(* PLC project Adressering.ecp, WAGO e!COCKPIT e!COCKPIT *)
(* stored: creationDateTime 2021-01-18T14:20:23.2110188, modificationDateTime 2021-01-18T11:51:27.6823754 *)

TYPE dtRomtype_112 : STRUCT
  RB601_V : BOOL;  (* Bevegelse *)
  RB601_HVAC : BOOL;  (* HVAC signal *)
  RT601_CT : REAL;  (* Rom temperatur *)
  RT602_CT : REAL;  (* Rom temperatur *)
  RT602_SP : REAL;  (* Temperatur SP *)
  RT601_SP_D : REAL;  (* Temperatur SP *)
  RT601_SP_S : REAL;  (* Temperatur SP standby *)
  RT601_SP_N : REAL;  (* Temperatur SP nattsenk *)
  RT601_SP_F : REAL;  (* Temperatur SP frostsikring *)
  RT601_CS : REAL;  (* Aktivt temperatur SP *)
  OPM : INT;  (* Rom modus *)
  OPM_CV : INT;  (* Rom modus verdi *)
END_STRUCT;
END_TYPE

TYPE dtRomtype_11102 : STRUCT
  RB601_V : BOOL;  (* Bevegelse *)
  RB601_HVAC : BOOL;  (* HVAC signal *)
  RT601_CT : REAL;  (* Rom temperatur *)
  RT601_SP_D : REAL;  (* Temperatur SP *)
  RT601_SP_S : REAL;  (* Temperatur SP standby *)
  RT601_SP_N : REAL;  (* Temperatur SP nattsenk *)
  RT601_SP_F : REAL;  (* Temperatur SP frostsikring *)
  RT601_CS : REAL;  (* Aktivt temperatur SP *)
  OPM : INT;  (* Rom modus *)
  OPM_CV : INT;  (* Rom modus verdi *)
  LH601_OP : REAL;  (* Varmepaadrag *)
  LH602_OP : REAL;  (* Varmepaadrag *)
  LH601_MAN : BOOL;  (* Force LH *)
END_STRUCT;
END_TYPE

TYPE dtRomtype_22111 : STRUCT
  RB601_V : BOOL;  (* Bevegelse *)
  RB602_V : BOOL;  (* Bevegelse *)
  RB601_HVAC : BOOL;  (* HVAC signal *)
  RB602_HVAC : BOOL;  (* HVAC signal *)
  RT601_CT : REAL;  (* Rom temperatur *)
  RT601_SP_D : REAL;  (* Temperatur SP *)
  RT601_SP_S : REAL;  (* Temperatur SP standby *)
  RT601_SP_N : REAL;  (* Temperatur SP nattsenk *)
  RT601_SP_F : REAL;  (* Temperatur SP frostsikring *)
  RT601_CS : REAL;  (* Aktivt temperatur SP *)
  OPM : INT;  (* Rom modus *)
  OPM_CV : INT;  (* Rom modus verdi *)
  RY601_CV : REAL;  (* Co2 Nivaa *)
  RY601_SP : REAL;  (* Co2 SP *)
  RY601_OP : REAL;  (* Co2 paadrag *)
  LH601_OP : REAL;  (* Varmepaadrag *)
  LH601_MAN : BOOL;  (* Force LH *)
END_STRUCT;
END_TYPE

TYPE dtRomtype_2211111 : STRUCT
  RB601_V : BOOL;  (* Bevegelse *)
  RB602_V : BOOL;  (* Bevegelse *)
  RB601_HVAC : BOOL;  (* HVAC signal *)
  RB602_HVAC : BOOL;  (* HVAC signal *)
  RT601_CT : REAL;  (* Rom temperatur *)
  RT601_SP_D : REAL;  (* Temperatur SP *)
  RT601_SP_S : REAL;  (* Temperatur SP standby *)
  RT601_SP_N : REAL;  (* Temperatur SP nattsenk *)
  RT601_SP_F : REAL;  (* Temperatur SP frostsikring *)
  RT601_CS : REAL;  (* Aktivt temperatur SP *)
  OPM : INT;  (* Rom modus *)
  OPM_CV : INT;  (* Rom modus verdi *)
  RY601_CV : REAL;  (* Co2 Nivaa *)
  RY601_SP : REAL;  (* Co2 SP *)
  RY601_OP : REAL;  (* Co2 paadrag *)
  LH601_OP : REAL;  (* Varmepaadrag *)
  LH601_MAN : BOOL;  (* Force LH *)
  LH601_CMD : BOOL;  (* LH601_CMD *)
  LC601_OP : REAL;  (* LC601_OP *)
  LC601_MAN : BOOL;  (* Force LC *)
END_STRUCT;
END_TYPE

TYPE dtRomtype_11111111 : STRUCT
  RB601_V : BOOL;  (* Bevegelse *)
  RB601_HVAC : BOOL;  (* HVAC signal *)
  RT601_CT : REAL;  (* Rom temperatur *)
  RT601_SP_D : REAL;  (* Temperatur SP *)
  RT601_SP_S : REAL;  (* Temperatur SP standby *)
  RT601_SP_N : REAL;  (* Temperatur SP nattsenk *)
  RT601_SP_F : REAL;  (* Temperatur SP frostsikring *)
  RT601_CS : REAL;  (* Aktivt temperatur SP *)
  OPM : INT;  (* Rom modus *)
  OPM_CV : INT;  (* Rom modus verdi *)
  RY601_CV : REAL;  (* Co2 Nivaa *)
  RY601_SP : REAL;  (* Co2 SP *)
  RY601_OP : REAL;  (* Co2 paadrag *)
  LH601_OP : REAL;  (* Varmepaadrag *)
  LH601_MAN : BOOL;  (* Force LH *)
  LH601_CMD : BOOL;  (* LH601_CMD *)
  LC601_OP : REAL;  (* LC601_OP *)
  LC601_MAN : BOOL;  (* Force LC *)
  LC601_CMD : BOOL;  (* LC601_CMD *)
END_STRUCT;
END_TYPE

TYPE dtRomtype_111111111 : STRUCT
  RB601_V : BOOL;  (* Bevegelse *)
  RB601_HVAC : BOOL;  (* HVAC signal *)
  RT601_CT : REAL;  (* Rom temperatur *)
  RT601_SP_D : REAL;  (* Temperatur SP *)
  RT601_SP_S : REAL;  (* Temperatur SP standby *)
  RT601_SP_N : REAL;  (* Temperatur SP nattsenk *)
  RT601_SP_F : REAL;  (* Temperatur SP frostsikring *)
  RT601_CS : REAL;  (* Aktivt temperatur SP *)
  OPM : INT;  (* Rom modus *)
  OPM_CV : INT;  (* Rom modus verdi *)
  RY601_CV : REAL;  (* Co2 Nivaa *)
  RY601_SP : REAL;  (* Co2 SP *)
  RY601_OP : REAL;  (* Co2 paadrag *)
  LH601_OP : REAL;  (* Varmepaadrag *)
  LH601_MAN : BOOL;  (* Force LH *)
  LH601_CMD : BOOL;  (* LH601_CMD *)
  LC601_OP : REAL;  (* LC601_OP *)
  LC601_MAN : BOOL;  (* Force LC *)
  LC601_CMD : BOOL;  (* LC601_CMD *)
  RT601_SP : REAL;  (* Temperatur SP feedback *)
END_STRUCT;
END_TYPE

TYPE dtRomtype_1111111111 : STRUCT
  RB601_V : BOOL;  (* Bevegelse *)
  RB601_HVAC : BOOL;  (* HVAC signal *)
  RT601_CT : REAL;  (* Rom temperatur *)
  RT601_SP_D : REAL;  (* Temperatur SP *)
  RT601_SP_S : REAL;  (* Temperatur SP standby *)
  RT601_SP_N : REAL;  (* Temperatur SP nattsenk *)
  RT601_SP_F : REAL;  (* Temperatur SP frostsikring *)
  RT601_CS : REAL;  (* Aktivt temperatur SP *)
  OPM : INT;  (* Rom modus *)
  OPM_CV : INT;  (* Rom modus verdi *)
  RY601_CV : REAL;  (* Co2 Nivaa *)
  RY601_SP : REAL;  (* Co2 SP *)
  RY601_OP : REAL;  (* Co2 paadrag *)
  LH601_OP : REAL;  (* Varmepaadrag *)
  LH601_MAN : BOOL;  (* Force LH *)
  LH601_CMD : BOOL;  (* LH601_CMD *)
  LC601_OP : REAL;  (* LC601_OP *)
  LC601_MAN : BOOL;  (* Force LC *)
  LC601_CMD : BOOL;  (* LC601_CMD *)
  RT601_SP : REAL;  (* Temperatur SP feedback *)
  RT601_SP_FB : REAL;  (* Temperatur SP *)
  RT601_SP_IN : REAL;  (* Temperatur SP lokalt panel *)
END_STRUCT;
END_TYPE

TYPE dtRomtype_11111111111 : STRUCT
  RB601_V : BOOL;  (* Bevegelse *)
  RB601_HVAC : BOOL;  (* HVAC signal *)
  RT601_CT : REAL;  (* Rom temperatur *)
  RT601_SP_D : REAL;  (* Temperatur SP *)
  RT601_SP_S : REAL;  (* Temperatur SP standby *)
  RT601_SP_N : REAL;  (* Temperatur SP nattsenk *)
  RT601_SP_F : REAL;  (* Temperatur SP frostsikring *)
  RT601_CS : REAL;  (* Aktivt temperatur SP *)
  OPM : INT;  (* Rom modus *)
  OPM_CV : INT;  (* Rom modus verdi *)
  RY601_CV : REAL;  (* Co2 Nivaa *)
  RY601_SP : REAL;  (* Co2 SP *)
  RY601_OP : REAL;  (* Co2 paadrag *)
  LH601_OP : REAL;  (* Varmepaadrag *)
  LH601_MAN : BOOL;  (* Force LH *)
  LH601_CMD : BOOL;  (* LH601_CMD *)
  LC601_OP : REAL;  (* LC601_OP *)
  LC601_MAN : BOOL;  (* Force LC *)
  LC601_CMD : BOOL;  (* LC601_CMD *)
  RT601_SP : REAL;  (* Temperatur SP feedback *)
  RT601_SP_FB : REAL;  (* Temperatur SP *)
  RT601_SP_IN : REAL;  (* Temperatur SP lokalt panel *)
  LU601_V : BOOL;  (* Befukter status *)
END_STRUCT;
END_TYPE

TYPE dtRomtype_111111111111 : STRUCT
  RB601_V : BOOL;  (* Bevegelse *)
  RB601_HVAC : BOOL;  (* HVAC signal *)
  RT601_CT : REAL;  (* Rom temperatur *)
  RT601_SP_D : REAL;  (* Temperatur SP *)
  RT601_SP_S : REAL;  (* Temperatur SP standby *)
  RT601_SP_N : REAL;  (* Temperatur SP nattsenk *)
  RT601_SP_F : REAL;  (* Temperatur SP frostsikring *)
  RT601_CS : REAL;  (* Aktivt temperatur SP *)
  OPM : INT;  (* Rom modus *)
  OPM_CV : INT;  (* Rom modus verdi *)
  RY601_CV : REAL;  (* Co2 Nivaa *)
  RY601_SP : REAL;  (* Co2 SP *)
  RY601_OP : REAL;  (* Co2 paadrag *)
  LH601_OP : REAL;  (* Varmepaadrag *)
  LH601_MAN : BOOL;  (* Force LH *)
  LH601_CMD : BOOL;  (* LH601_CMD *)
  LC601_OP : REAL;  (* LC601_OP *)
  LC601_MAN : BOOL;  (* Force LC *)
  LC601_CMD : BOOL;  (* LC601_CMD *)
  RT601_SP : REAL;  (* Temperatur SP feedback *)
  RT601_SP_FB : REAL;  (* Temperatur SP *)
  RT601_SP_IN : REAL;  (* Temperatur SP lokalt panel *)
  LU601_V : BOOL;  (* Befukter status *)
  LU601_AL : BOOL;  (* Befukter alarm/feil *)
END_STRUCT;
END_TYPE

TYPE dtRomtype_1111111111111 : STRUCT
  RB601_V : BOOL;  (* Bevegelse *)
  RB601_HVAC : BOOL;  (* HVAC signal *)
  RT601_CT : REAL;  (* Rom temperatur *)
  RT601_SP_D : REAL;  (* Temperatur SP *)
  RT601_SP_S : REAL;  (* Temperatur SP standby *)
  RT601_SP_N : REAL;  (* Temperatur SP nattsenk *)
  RT601_SP_F : REAL;  (* Temperatur SP frostsikring *)
  RT601_CS : REAL;  (* Aktivt temperatur SP *)
  OPM : INT;  (* Rom modus *)
  OPM_CV : INT;  (* Rom modus verdi *)
  RY601_CV : REAL;  (* Co2 Nivaa *)
  RY601_SP : REAL;  (* Co2 SP *)
  RY601_OP : REAL;  (* Co2 paadrag *)
  LH601_OP : REAL;  (* Varmepaadrag *)
  LH601_MAN : BOOL;  (* Force LH *)
  LH601_CMD : BOOL;  (* LH601_CMD *)
  LC601_OP : REAL;  (* LC601_OP *)
  LC601_MAN : BOOL;  (* Force LC *)
  LC601_CMD : BOOL;  (* LC601_CMD *)
  RT601_SP : REAL;  (* Temperatur SP feedback *)
  RT601_SP_FB : REAL;  (* Temperatur SP *)
  RT601_SP_IN : REAL;  (* Temperatur SP lokalt panel *)
  LU601_V : BOOL;  (* Befukter status *)
  LU601_AL : BOOL;  (* Befukter alarm/feil *)
  LU601_CMD : BOOL;  (* Befukter tillat start *)
END_STRUCT;
END_TYPE

TYPE dtRomtype_2222222222222 : STRUCT
  RB601_V : BOOL;  (* Bevegelse *)
  RB602_V : BOOL;  (* Bevegelse *)
  RB601_HVAC : BOOL;  (* HVAC signal *)
  RB602_HVAC : BOOL;  (* HVAC signal *)
  RT601_CT : REAL;  (* Rom temperatur *)
  RT602_CT : REAL;  (* Rom temperatur *)
  RT602_SP : REAL;  (* Temperatur SP *)
  RT601_SP_D : REAL;  (* Temperatur SP *)
  RT601_SP_S : REAL;  (* Temperatur SP standby *)
  RT601_SP_N : REAL;  (* Temperatur SP nattsenk *)
  RT601_SP_F : REAL;  (* Temperatur SP frostsikring *)
  RT601_CS : REAL;  (* Aktivt temperatur SP *)
  OPM : INT;  (* Rom modus *)
  OPM_CV : INT;  (* Rom modus verdi *)
  RY601_CV : REAL;  (* Co2 Nivaa *)
  RY602_CV : REAL;  (* Co2 Nivaa *)
  RY601_SP : REAL;  (* Co2 SP *)
  RY601_OP : REAL;  (* Co2 paadrag *)
  LH601_OP : REAL;  (* Varmepaadrag *)
  LH602_OP : REAL;  (* Varmepaadrag *)
  LH601_MAN : BOOL;  (* Force LH *)
  LH601_CMD : BOOL;  (* LH601_CMD *)
  LH602_CMD : BOOL;  (* LH602_CMD *)
  LC601_OP : REAL;  (* LC601_OP *)
  LC602_OP : REAL;  (* LC602_OP *)
  LC601_MAN : BOOL;  (* Force LC *)
  LC601_CMD : BOOL;  (* LC601_CMD *)
  LC602_CMD : BOOL;  (* LC602_CMD *)
  RT601_SP : REAL;  (* Temperatur SP feedback *)
  RT601_SP_FB : REAL;  (* Temperatur SP *)
  RT601_SP_IN : REAL;  (* Temperatur SP lokalt panel *)
  RT602_SP_FB : REAL;  (* Temperatur SP *)
  RT602_SP_IN : REAL;  (* Temperatur SP lokalt panel *)
  LU601_V : BOOL;  (* Befukter status *)
  LU602_V : BOOL;  (* Befukter status *)
  LU601_AL : BOOL;  (* Befukter alarm/feil *)
  LU602_AL : BOOL;  (* Befukter alarm/feil *)
  LU601_CMD : BOOL;  (* Befukter tillat start *)
  LU602_CMD : BOOL;  (* Befukter tillat start *)
END_STRUCT;
END_TYPE

{attribute 'qualified_only'}
VAR_GLOBAL  (* STLV80_563 *)
  STLV80_A_563_KNX_Card_1_Status : BOOL;  (* KNX kort 1 status *)
  STLV80_A_563_5A201 : dtRomtype_112;
  STLV80_A_563_5A202 : dtRomtype_11102;
  STLV80_A_563_5A203 : dtRomtype_22111;
  STLV80_A_563_5A301 : dtRomtype_2211111;
  STLV80_A_563_5A302 : dtRomtype_11111111;
  STLV80_A_563_5B201 : dtRomtype_111111111;
  STLV80_A_563_5B202 : dtRomtype_1111111111;
  STLV80_A_563_5B301 : dtRomtype_11111111111;
  STLV80_A_563_5B302 : dtRomtype_111111111111;
  STLV80_A_563_5C201 : dtRomtype_1111111111111;
  STLV80_A_563_5C202 : dtRomtype_2222222222222;
END_VAR

FUNCTION_BLOCK fbRomtype_112
  VAR_INPUT
    RB601_HVAC : BOOL;
    RT601_CT : REAL;
    RT602_CT : REAL;
    RT602_SP : REAL;
    RT601_SP_D : REAL;
    RT601_SP_S : REAL;
    RT601_SP_N : REAL;
    RT601_SP_F : REAL;
    OPM : INT;
  END_VAR
  VAR_OUTPUT
    OPM_CV : INT;
    RT601_CS : REAL;
    RT602_CS : REAL;
  END_VAR

(* CFC diagram, written out as Structured Text *)
END_FUNCTION_BLOCK

FUNCTION_BLOCK fbRomtype_11102
  VAR_INPUT
    RB601_HVAC : BOOL;
    RT601_CT : REAL;
    RT601_SP_D : REAL;
    RT601_SP_S : REAL;
    RT601_SP_N : REAL;
    RT601_SP_F : REAL;
    OPM : INT;
    LH601_MAN : BOOL;
  END_VAR
  VAR_OUTPUT
    OPM_CV : INT;
    RT601_CS : REAL;
    LH601_OP : REAL;
    LH602_OP : REAL;
  END_VAR

(* CFC diagram, written out as Structured Text *)
END_FUNCTION_BLOCK

FUNCTION_BLOCK fbRomtype_22111
  VAR_INPUT
    RB601_HVAC : BOOL;
    RB602_HVAC : BOOL;
    RT601_CT : REAL;
    RT601_SP_D : REAL;
    RT601_SP_S : REAL;
    RT601_SP_N : REAL;
    RT601_SP_F : REAL;
    OPM : INT;
    RY601_CV : REAL;
    RY601_SP : REAL;
    LH601_MAN : BOOL;
  END_VAR
  VAR_OUTPUT
    OPM_CV : INT;
    RT601_CS : REAL;
    RY601_OP : REAL;
    LH601_OP : REAL;
  END_VAR

(* CFC diagram, written out as Structured Text *)
END_FUNCTION_BLOCK

FUNCTION_BLOCK fbRomtype_2211111
  VAR_INPUT
    RB601_HVAC : BOOL;
    RB602_HVAC : BOOL;
    RT601_CT : REAL;
    RT601_SP_D : REAL;
    RT601_SP_S : REAL;
    RT601_SP_N : REAL;
    RT601_SP_F : REAL;
    OPM : INT;
    RY601_CV : REAL;
    RY601_SP : REAL;
    LH601_MAN : BOOL;
    LC601_MAN : BOOL;
  END_VAR
  VAR_OUTPUT
    OPM_CV : INT;
    RT601_CS : REAL;
    RY601_OP : REAL;
    LH601_OP : REAL;
    LH601_CMD : BOOL;
    LC601_OP : REAL;
  END_VAR

(* CFC diagram, written out as Structured Text *)
END_FUNCTION_BLOCK

FUNCTION_BLOCK fbRomtype_11111111
  VAR_INPUT
    RB601_HVAC : BOOL;
    RT601_CT : REAL;
    RT601_SP_D : REAL;
    RT601_SP_S : REAL;
    RT601_SP_N : REAL;
    RT601_SP_F : REAL;
    OPM : INT;
    RY601_CV : REAL;
    RY601_SP : REAL;
    LH601_MAN : BOOL;
    LC601_MAN : BOOL;
  END_VAR
  VAR_OUTPUT
    OPM_CV : INT;
    RT601_CS : REAL;
    RY601_OP : REAL;
    LH601_OP : REAL;
    LH601_CMD : BOOL;
    LC601_OP : REAL;
    LC601_CMD : BOOL;
  END_VAR

(* CFC diagram, written out as Structured Text *)
END_FUNCTION_BLOCK

FUNCTION_BLOCK fbRomtype_111111111
  VAR_INPUT
    RB601_HVAC : BOOL;
    RT601_CT : REAL;
    RT601_SP_D : REAL;
    RT601_SP_S : REAL;
    RT601_SP_N : REAL;
    RT601_SP_F : REAL;
    OPM : INT;
    RY601_CV : REAL;
    RY601_SP : REAL;
    LH601_MAN : BOOL;
    LC601_MAN : BOOL;
    RT601_SP_IN : REAL;
  END_VAR
  VAR_OUTPUT
    OPM_CV : INT;
    RT601_CS : REAL;
    RY601_OP : REAL;
    LH601_OP : REAL;
    LH601_CMD : BOOL;
    LC601_OP : REAL;
    LC601_CMD : BOOL;
  END_VAR

(* CFC diagram, written out as Structured Text *)
END_FUNCTION_BLOCK

FUNCTION_BLOCK fbRomtype_1111111111
  VAR_INPUT
    RB601_HVAC : BOOL;
    RT601_CT : REAL;
    RT601_SP_D : REAL;
    RT601_SP_S : REAL;
    RT601_SP_N : REAL;
    RT601_SP_F : REAL;
    OPM : INT;
    RY601_CV : REAL;
    RY601_SP : REAL;
    LH601_MAN : BOOL;
    LC601_MAN : BOOL;
    RT601_SP_IN : REAL;
  END_VAR
  VAR_OUTPUT
    OPM_CV : INT;
    RT601_CS : REAL;
    RY601_OP : REAL;
    LH601_OP : REAL;
    LH601_CMD : BOOL;
    LC601_OP : REAL;
    LC601_CMD : BOOL;
  END_VAR

(* CFC diagram, written out as Structured Text *)
END_FUNCTION_BLOCK

FUNCTION_BLOCK fbRomtype_11111111111
  VAR_INPUT
    RB601_HVAC : BOOL;
    RT601_CT : REAL;
    RT601_SP_D : REAL;
    RT601_SP_S : REAL;
    RT601_SP_N : REAL;
    RT601_SP_F : REAL;
    OPM : INT;
    RY601_CV : REAL;
    RY601_SP : REAL;
    LH601_MAN : BOOL;
    LC601_MAN : BOOL;
    RT601_SP_IN : REAL;
    LU601_V : BOOL;
  END_VAR
  VAR_OUTPUT
    OPM_CV : INT;
    RT601_CS : REAL;
    RY601_OP : REAL;
    LH601_OP : REAL;
    LH601_CMD : BOOL;
    LC601_OP : REAL;
    LC601_CMD : BOOL;
  END_VAR

(* CFC diagram, written out as Structured Text *)
END_FUNCTION_BLOCK

FUNCTION_BLOCK fbRomtype_111111111111
  VAR_INPUT
    RB601_HVAC : BOOL;
    RT601_CT : REAL;
    RT601_SP_D : REAL;
    RT601_SP_S : REAL;
    RT601_SP_N : REAL;
    RT601_SP_F : REAL;
    OPM : INT;
    RY601_CV : REAL;
    RY601_SP : REAL;
    LH601_MAN : BOOL;
    LC601_MAN : BOOL;
    RT601_SP_IN : REAL;
    LU601_V : BOOL;
    LU601_AL : BOOL;
  END_VAR
  VAR_OUTPUT
    OPM_CV : INT;
    RT601_CS : REAL;
    RY601_OP : REAL;
    LH601_OP : REAL;
    LH601_CMD : BOOL;
    LC601_OP : REAL;
    LC601_CMD : BOOL;
  END_VAR

(* CFC diagram, written out as Structured Text *)
END_FUNCTION_BLOCK

FUNCTION_BLOCK fbRomtype_1111111111111
  VAR_INPUT
    RB601_HVAC : BOOL;
    RT601_CT : REAL;
    RT601_SP_D : REAL;
    RT601_SP_S : REAL;
    RT601_SP_N : REAL;
    RT601_SP_F : REAL;
    OPM : INT;
    RY601_CV : REAL;
    RY601_SP : REAL;
    LH601_MAN : BOOL;
    LC601_MAN : BOOL;
    RT601_SP_IN : REAL;
    LU601_V : BOOL;
    LU601_AL : BOOL;
  END_VAR
  VAR_OUTPUT
    OPM_CV : INT;
    RT601_CS : REAL;
    RY601_OP : REAL;
    LH601_OP : REAL;
    LH601_CMD : BOOL;
    LC601_OP : REAL;
    LC601_CMD : BOOL;
    LU601_CMD : BOOL;
  END_VAR

(* CFC diagram, written out as Structured Text *)
END_FUNCTION_BLOCK

FUNCTION_BLOCK fbRomtype_2222222222222
  VAR_INPUT
    RB601_HVAC : BOOL;
    RB602_HVAC : BOOL;
    RT601_CT : REAL;
    RT602_CT : REAL;
    RT602_SP : REAL;
    RT601_SP_D : REAL;
    RT601_SP_S : REAL;
    RT601_SP_N : REAL;
    RT601_SP_F : REAL;
    OPM : INT;
    RY601_CV : REAL;
    RY602_CV : REAL;
    RY601_SP : REAL;
    LH601_MAN : BOOL;
    LC601_MAN : BOOL;
    RT601_SP_IN : REAL;
    RT602_SP_IN : REAL;
    LU601_V : BOOL;
    LU602_V : BOOL;
    LU601_AL : BOOL;
    LU602_AL : BOOL;
  END_VAR
  VAR_OUTPUT
    OPM_CV : INT;
    RT601_CS : REAL;
    RT602_CS : REAL;
    RY601_OP : REAL;
    LH601_OP : REAL;
    LH602_OP : REAL;
    LH601_CMD : BOOL;
    LH602_CMD : BOOL;
    LC601_OP : REAL;
    LC602_OP : REAL;
    LC601_CMD : BOOL;
    LC602_CMD : BOOL;
    LU601_CMD : BOOL;
    LU602_CMD : BOOL;
  END_VAR

(* CFC diagram, written out as Structured Text *)
END_FUNCTION_BLOCK

PROGRAM PRG_563_KNX_1
  VAR
    i : INT := 0;  (* Felles *)
    Interval : OSCAT_BASIC.CLK_PRG;
    typDPT : typDPT;
    KNX_master_1 : WagoAppKNX.FbKNX_Master;  (* Master *)
    M1_001_5A201_RB601_V : fbDPT_Switch_pro;  (* 5A201 *)
    M1_002_5A201_RB601_HVAC : fbDPT_Switch_pro;
    M1_003_5A201_RT601_CT : fbDPT_Value_Temp_pro;
    M1_004_5A201_RT602_CT : fbDPT_Value_Temp_pro;
    M1_005_5A202_RB601_V : fbDPT_Switch_pro;  (* 5A202 *)
    M1_006_5A202_RB601_HVAC : fbDPT_Switch_pro;
    M1_007_5A202_RT601_CT : fbDPT_Value_Temp_pro;
    M1_008_5A203_RB601_V : fbDPT_Switch_pro;  (* 5A203 *)
    M1_009_5A203_RB602_V : fbDPT_Switch_pro;
    M1_010_5A203_RB601_HVAC : fbDPT_Switch_pro;
    M1_011_5A203_RT601_CT : fbDPT_Value_Temp_pro;
    M1_012_5A203_RY601_CV : fbDPT_Value_AirQuality_pro;
    M1_013_5A301_RB601_V : fbDPT_Switch_pro;  (* 5A301 *)
    M1_014_5A301_RB602_V : fbDPT_Switch_pro;
    M1_015_5A301_RB601_HVAC : fbDPT_Switch_pro;
    M1_016_5A301_RB602_HVAC : fbDPT_Switch_pro;
    M1_017_5A301_RT601_CT : fbDPT_Value_Temp_pro;
    M1_018_5A301_RY601_CV : fbDPT_Value_AirQuality_pro;
    M1_019_5A301_LH601_OP : fbDPT_Scaling_pro;
    M1_020_5A302_RB601_V : fbDPT_Switch_pro;  (* 5A302 *)
    M1_021_5A302_RB601_HVAC : fbDPT_Switch_pro;
    M1_022_5A302_RT601_CT : fbDPT_Value_Temp_pro;
    M1_023_5A302_RY601_CV : fbDPT_Value_AirQuality_pro;
    M1_024_5A302_LH601_OP : fbDPT_Scaling_pro;
    M1_025_5A302_LH601_CMD : fbDPT_Switch_pro;
    M1_026_5A302_LC601_OP : fbDPT_Scaling_pro;
    M1_027_5A302_LC601_CMD : fbDPT_Switch_pro;
    M1_028_5B201_RB601_V : fbDPT_Switch_pro;  (* 5B201 *)
    M1_029_5B201_RB601_HVAC : fbDPT_Switch_pro;
    M1_030_5B201_RT601_CT : fbDPT_Value_Temp_pro;
    M1_031_5B201_RY601_CV : fbDPT_Value_AirQuality_pro;
    M1_032_5B201_LH601_OP : fbDPT_Scaling_pro;
    M1_033_5B201_LH601_CMD : fbDPT_Switch_pro;
    M1_034_5B201_LC601_OP : fbDPT_Scaling_pro;
    M1_035_5B201_LC601_CMD : fbDPT_Switch_pro;
    M1_036_5B201_RT601_SP : fbDPT_Value_Temp_pro;
    M1_037_5B202_RB601_V : fbDPT_Switch_pro;  (* 5B202 *)
    M1_038_5B202_RB601_HVAC : fbDPT_Switch_pro;
    M1_039_5B202_RT601_CT : fbDPT_Value_Temp_pro;
    M1_040_5B202_RY601_CV : fbDPT_Value_AirQuality_pro;
    M1_041_5B202_LH601_OP : fbDPT_Scaling_pro;
    M1_042_5B202_LH601_CMD : fbDPT_Switch_pro;
    M1_043_5B202_LC601_OP : fbDPT_Scaling_pro;
    M1_044_5B202_LC601_CMD : fbDPT_Switch_pro;
    M1_045_5B202_RT601_SP : fbDPT_Value_Temp_pro;
    M1_046_5B202_RT601_SP_FB : fbDPT_Value_Temp_pro;
    M1_047_5B301_RB601_V : fbDPT_Switch_pro;  (* 5B301 *)
    M1_048_5B301_RB601_HVAC : fbDPT_Switch_pro;
    M1_049_5B301_RT601_CT : fbDPT_Value_Temp_pro;
    M1_050_5B301_RY601_CV : fbDPT_Value_AirQuality_pro;
    M1_051_5B301_LH601_OP : fbDPT_Scaling_pro;
    M1_052_5B301_LH601_CMD : fbDPT_Switch_pro;
    M1_053_5B301_LC601_OP : fbDPT_Scaling_pro;
    M1_054_5B301_LC601_CMD : fbDPT_Switch_pro;
    M1_055_5B301_RT601_SP : fbDPT_Value_Temp_pro;
    M1_056_5B301_RT601_SP_FB : fbDPT_Value_Temp_pro;
    M1_057_5B301_LU601_V : fbDPT_Switch_pro;
    M1_058_5B302_RB601_V : fbDPT_Switch_pro;  (* 5B302 *)
    M1_059_5B302_RB601_HVAC : fbDPT_Switch_pro;
    M1_060_5B302_RT601_CT : fbDPT_Value_Temp_pro;
    M1_061_5B302_RY601_CV : fbDPT_Value_AirQuality_pro;
    M1_062_5B302_LH601_OP : fbDPT_Scaling_pro;
    M1_063_5B302_LH601_CMD : fbDPT_Switch_pro;
    M1_064_5B302_LC601_OP : fbDPT_Scaling_pro;
    M1_065_5B302_LC601_CMD : fbDPT_Switch_pro;
    M1_066_5B302_RT601_SP : fbDPT_Value_Temp_pro;
    M1_067_5B302_RT601_SP_FB : fbDPT_Value_Temp_pro;
    M1_068_5B302_LU601_V : fbDPT_Switch_pro;
    M1_069_5B302_LU601_AL : fbDPT_Switch_pro;
    M1_070_5C201_RB601_V : fbDPT_Switch_pro;  (* 5C201 *)
    M1_071_5C201_RB601_HVAC : fbDPT_Switch_pro;
    M1_072_5C201_RT601_CT : fbDPT_Value_Temp_pro;
    M1_073_5C201_RY601_CV : fbDPT_Value_AirQuality_pro;
    M1_074_5C201_LH601_OP : fbDPT_Scaling_pro;
    M1_075_5C201_LH601_CMD : fbDPT_Switch_pro;
    M1_076_5C201_LC601_OP : fbDPT_Scaling_pro;
    M1_077_5C201_LC601_CMD : fbDPT_Switch_pro;
    M1_078_5C201_RT601_SP : fbDPT_Value_Temp_pro;
    M1_079_5C201_RT601_SP_FB : fbDPT_Value_Temp_pro;
    M1_080_5C201_LU601_V : fbDPT_Switch_pro;
    M1_081_5C201_LU601_AL : fbDPT_Switch_pro;
    M1_082_5C201_LU601_CMD : fbDPT_Switch_pro;
    M1_083_5C202_RB601_V : fbDPT_Switch_pro;  (* 5C202 *)
    M1_084_5C202_RB602_V : fbDPT_Switch_pro;
    M1_085_5C202_RB601_HVAC : fbDPT_Switch_pro;
    M1_086_5C202_RB602_HVAC : fbDPT_Switch_pro;
    M1_087_5C202_RT601_CT : fbDPT_Value_Temp_pro;
    M1_088_5C202_RT602_CT : fbDPT_Value_Temp_pro;
    M1_089_5C202_RY601_CV : fbDPT_Value_AirQuality_pro;
    M1_090_5C202_RY602_CV : fbDPT_Value_AirQuality_pro;
    M1_091_5C202_LH601_OP : fbDPT_Scaling_pro;
    M1_092_5C202_LH602_OP : fbDPT_Scaling_pro;
    M1_093_5C202_LH601_CMD : fbDPT_Switch_pro;
    M1_094_5C202_LH602_CMD : fbDPT_Switch_pro;
    M1_095_5C202_LC601_OP : fbDPT_Scaling_pro;
    M1_096_5C202_LC602_OP : fbDPT_Scaling_pro;
    M1_097_5C202_LC601_CMD : fbDPT_Switch_pro;
    M1_098_5C202_LC602_CMD : fbDPT_Switch_pro;
    M1_099_5C202_RT601_SP : fbDPT_Value_Temp_pro;
    M1_0100_5C202_RT602_SP : fbDPT_Value_Temp_pro;
    M1_101_5C202_RT601_SP_FB : fbDPT_Value_Temp_pro;
    M1_102_5C202_RT602_SP_FB : fbDPT_Value_Temp_pro;
    M1_103_5C202_LU601_V : fbDPT_Switch_pro;
    M1_104_5C202_LU602_V : fbDPT_Switch_pro;
    M1_105_5C202_LU601_AL : fbDPT_Switch_pro;
    M1_106_5C202_LU602_AL : fbDPT_Switch_pro;
    M1_107_5C202_LU601_CMD : fbDPT_Switch_pro;
    M1_108_5C202_LU602_CMD : fbDPT_Switch_pro;
  END_VAR
  VAR  (* added by the conversion: wires and edge detectors of the diagram *)
    _ADD9_OUT : INT;
    _GT15_OUT : BOOL;
    _MOVE19_ENO : BOOL;
    _MOVE19_OUT : INT;
  END_VAR

(* CFC diagram, written out as Structured Text *)
(* KNX Sending interval *)
(* KNX Master *)
Interval(PT := t#2M);
_ADD9_OUT := BOOL_TO_INT(Interval.Q) + i;
i := _ADD9_OUT;
_GT15_OUT := i > 30;
_MOVE19_OUT := MOVE(EN := _GT15_OUT, IN := 0, ENO => _MOVE19_ENO);
IF _MOVE19_ENO THEN i := _MOVE19_OUT; END_IF;
KNX_master_1(I_Port := IoConfig_Globals.KNX_EIB_TP1_Interface, bPortKNX := 1);
STLV80_563.STLV80_A_563_KNX_Card_1_Status := KNX_master_1.sStatus = 'OK';
(* Rom 5A201 *)
(* RB601_V *)
(* RB601_HVAC *)
M1_001_5A201_RB601_V(bPortKNX := 1, dwIndex_DPT := 1, typDPT := typDPT);
STLV80_563.STLV80_A_563_5A201.RB601_V := M1_001_5A201_RB601_V.xSwitch_OUT;
M1_002_5A201_RB601_HVAC(bPortKNX := 1, dwIndex_DPT := 2, typDPT := typDPT);
STLV80_563.STLV80_A_563_5A201.RB601_HVAC := M1_002_5A201_RB601_HVAC.xSwitch_OUT;
(* RT601_CT *)
(* RT602_CT *)
M1_003_5A201_RT601_CT(bPortKNX := 1, dwIndex_DPT := 3, typDPT := typDPT);
STLV80_563.STLV80_A_563_5A201.RT601_CT := M1_003_5A201_RT601_CT.rValue_OUT;
M1_004_5A201_RT602_CT(bPortKNX := 1, dwIndex_DPT := 4, typDPT := typDPT);
STLV80_563.STLV80_A_563_5A201.RT602_CT := M1_004_5A201_RT602_CT.rValue_OUT;
(* Rom 5A202 *)
(* RB601_V *)
(* RB601_HVAC *)
M1_005_5A202_RB601_V(bPortKNX := 1, dwIndex_DPT := 5, typDPT := typDPT);
STLV80_563.STLV80_A_563_5A202.RB601_V := M1_005_5A202_RB601_V.xSwitch_OUT;
M1_006_5A202_RB601_HVAC(bPortKNX := 1, dwIndex_DPT := 6, typDPT := typDPT);
STLV80_563.STLV80_A_563_5A202.RB601_HVAC := M1_006_5A202_RB601_HVAC.xSwitch_OUT;
(* RT601_CT *)
M1_007_5A202_RT601_CT(bPortKNX := 1, dwIndex_DPT := 7, typDPT := typDPT);
STLV80_563.STLV80_A_563_5A202.RT601_CT := M1_007_5A202_RT601_CT.rValue_OUT;
(* Rom 5A203 *)
(* RB601_V *)
(* RB602_V *)
M1_008_5A203_RB601_V(bPortKNX := 1, dwIndex_DPT := 8, typDPT := typDPT);
STLV80_563.STLV80_A_563_5A203.RB601_V := M1_008_5A203_RB601_V.xSwitch_OUT;
M1_009_5A203_RB602_V(bPortKNX := 1, dwIndex_DPT := 9, typDPT := typDPT);
STLV80_563.STLV80_A_563_5A203.RB602_V := M1_009_5A203_RB602_V.xSwitch_OUT;
(* RB601_HVAC *)
(* RT601_CT *)
M1_010_5A203_RB601_HVAC(bPortKNX := 1, dwIndex_DPT := 10, typDPT := typDPT);
STLV80_563.STLV80_A_563_5A203.RB601_HVAC := M1_010_5A203_RB601_HVAC.xSwitch_OUT;
M1_011_5A203_RT601_CT(bPortKNX := 1, dwIndex_DPT := 11, typDPT := typDPT);
STLV80_563.STLV80_A_563_5A203.RT601_CT := M1_011_5A203_RT601_CT.rValue_OUT;
(* RY601_CV *)
M1_012_5A203_RY601_CV(bPortKNX := 1, dwIndex_DPT := 12, typDPT := typDPT);
STLV80_563.STLV80_A_563_5A203.RY601_CV := M1_012_5A203_RY601_CV.rValue_OUT;
(* Rom 5A301 *)
(* RB601_V *)
(* RB602_V *)
M1_013_5A301_RB601_V(bPortKNX := 1, dwIndex_DPT := 13, typDPT := typDPT);
STLV80_563.STLV80_A_563_5A301.RB601_V := M1_013_5A301_RB601_V.xSwitch_OUT;
M1_014_5A301_RB602_V(bPortKNX := 1, dwIndex_DPT := 14, typDPT := typDPT);
STLV80_563.STLV80_A_563_5A301.RB602_V := M1_014_5A301_RB602_V.xSwitch_OUT;
(* RB601_HVAC *)
(* RB602_HVAC *)
M1_015_5A301_RB601_HVAC(bPortKNX := 1, dwIndex_DPT := 15, typDPT := typDPT);
STLV80_563.STLV80_A_563_5A301.RB601_HVAC := M1_015_5A301_RB601_HVAC.xSwitch_OUT;
M1_016_5A301_RB602_HVAC(bPortKNX := 1, dwIndex_DPT := 16, typDPT := typDPT);
STLV80_563.STLV80_A_563_5A301.RB602_HVAC := M1_016_5A301_RB602_HVAC.xSwitch_OUT;
(* RT601_CT *)
(* RY601_CV *)
M1_017_5A301_RT601_CT(bPortKNX := 1, dwIndex_DPT := 17, typDPT := typDPT);
STLV80_563.STLV80_A_563_5A301.RT601_CT := M1_017_5A301_RT601_CT.rValue_OUT;
M1_018_5A301_RY601_CV(bPortKNX := 1, dwIndex_DPT := 18, typDPT := typDPT);
STLV80_563.STLV80_A_563_5A301.RY601_CV := M1_018_5A301_RY601_CV.rValue_OUT;
(* LH601_OP *)
M1_019_5A301_LH601_OP(bPortKNX := 1, dwIndex_DPT := 19, rValue_IN := STLV80_563.STLV80_A_563_5A301.LH601_OP, xUpdate_KNX := i = 0, typDPT := typDPT);
(* Rom 5A302 *)
(* RB601_V *)
(* RB601_HVAC *)
M1_020_5A302_RB601_V(bPortKNX := 1, dwIndex_DPT := 20, typDPT := typDPT);
STLV80_563.STLV80_A_563_5A302.RB601_V := M1_020_5A302_RB601_V.xSwitch_OUT;
M1_021_5A302_RB601_HVAC(bPortKNX := 1, dwIndex_DPT := 21, typDPT := typDPT);
STLV80_563.STLV80_A_563_5A302.RB601_HVAC := M1_021_5A302_RB601_HVAC.xSwitch_OUT;
(* RT601_CT *)
(* RY601_CV *)
M1_022_5A302_RT601_CT(bPortKNX := 1, dwIndex_DPT := 22, typDPT := typDPT);
STLV80_563.STLV80_A_563_5A302.RT601_CT := M1_022_5A302_RT601_CT.rValue_OUT;
M1_023_5A302_RY601_CV(bPortKNX := 1, dwIndex_DPT := 23, typDPT := typDPT);
STLV80_563.STLV80_A_563_5A302.RY601_CV := M1_023_5A302_RY601_CV.rValue_OUT;
(* LH601_OP *)
(* LH601_CMD *)
M1_024_5A302_LH601_OP(bPortKNX := 1, dwIndex_DPT := 24, rValue_IN := STLV80_563.STLV80_A_563_5A302.LH601_OP, xUpdate_KNX := i = 1, typDPT := typDPT);
M1_025_5A302_LH601_CMD(bPortKNX := 1, dwIndex_DPT := 25, xSwitch_IN := STLV80_563.STLV80_A_563_5A302.LH601_CMD, xUpdate_KNX := i = 2, typDPT := typDPT);
(* LC601_OP *)
(* LC601_CMD *)
M1_026_5A302_LC601_OP(bPortKNX := 1, dwIndex_DPT := 26, rValue_IN := STLV80_563.STLV80_A_563_5A302.LC601_OP, xUpdate_KNX := i = 3, typDPT := typDPT);
M1_027_5A302_LC601_CMD(bPortKNX := 1, dwIndex_DPT := 27, xSwitch_IN := STLV80_563.STLV80_A_563_5A302.LC601_CMD, xUpdate_KNX := i = 4, typDPT := typDPT);
(* Rom 5B201 *)
(* RB601_V *)
(* RB601_HVAC *)
M1_028_5B201_RB601_V(bPortKNX := 1, dwIndex_DPT := 28, typDPT := typDPT);
STLV80_563.STLV80_A_563_5B201.RB601_V := M1_028_5B201_RB601_V.xSwitch_OUT;
M1_029_5B201_RB601_HVAC(bPortKNX := 1, dwIndex_DPT := 29, typDPT := typDPT);
STLV80_563.STLV80_A_563_5B201.RB601_HVAC := M1_029_5B201_RB601_HVAC.xSwitch_OUT;
(* RT601_CT *)
(* RY601_CV *)
M1_030_5B201_RT601_CT(bPortKNX := 1, dwIndex_DPT := 30, typDPT := typDPT);
STLV80_563.STLV80_A_563_5B201.RT601_CT := M1_030_5B201_RT601_CT.rValue_OUT;
M1_031_5B201_RY601_CV(bPortKNX := 1, dwIndex_DPT := 31, typDPT := typDPT);
STLV80_563.STLV80_A_563_5B201.RY601_CV := M1_031_5B201_RY601_CV.rValue_OUT;
(* LH601_OP *)
(* LH601_CMD *)
M1_032_5B201_LH601_OP(bPortKNX := 1, dwIndex_DPT := 32, rValue_IN := STLV80_563.STLV80_A_563_5B201.LH601_OP, xUpdate_KNX := i = 5, typDPT := typDPT);
M1_033_5B201_LH601_CMD(bPortKNX := 1, dwIndex_DPT := 33, xSwitch_IN := STLV80_563.STLV80_A_563_5B201.LH601_CMD, xUpdate_KNX := i = 6, typDPT := typDPT);
(* LC601_OP *)
(* LC601_CMD *)
M1_034_5B201_LC601_OP(bPortKNX := 1, dwIndex_DPT := 34, rValue_IN := STLV80_563.STLV80_A_563_5B201.LC601_OP, xUpdate_KNX := i = 7, typDPT := typDPT);
M1_035_5B201_LC601_CMD(bPortKNX := 1, dwIndex_DPT := 35, xSwitch_IN := STLV80_563.STLV80_A_563_5B201.LC601_CMD, xUpdate_KNX := i = 8, typDPT := typDPT);
(* RT601_SP *)
M1_036_5B201_RT601_SP(bPortKNX := 1, dwIndex_DPT := 36, rValue_IN := STLV80_563.STLV80_A_563_5B201.RT601_SP_D, xUpdate_KNX := NOT STLV80_563.STLV80_A_563_5B201.RB601_HVAC, typDPT := typDPT);
(* Rom 5B202 *)
(* RB601_V *)
(* RB601_HVAC *)
M1_037_5B202_RB601_V(bPortKNX := 1, dwIndex_DPT := 37, typDPT := typDPT);
STLV80_563.STLV80_A_563_5B202.RB601_V := M1_037_5B202_RB601_V.xSwitch_OUT;
M1_038_5B202_RB601_HVAC(bPortKNX := 1, dwIndex_DPT := 38, typDPT := typDPT);
STLV80_563.STLV80_A_563_5B202.RB601_HVAC := M1_038_5B202_RB601_HVAC.xSwitch_OUT;
(* RT601_CT *)
(* RY601_CV *)
M1_039_5B202_RT601_CT(bPortKNX := 1, dwIndex_DPT := 39, typDPT := typDPT);
STLV80_563.STLV80_A_563_5B202.RT601_CT := M1_039_5B202_RT601_CT.rValue_OUT;
M1_040_5B202_RY601_CV(bPortKNX := 1, dwIndex_DPT := 40, typDPT := typDPT);
STLV80_563.STLV80_A_563_5B202.RY601_CV := M1_040_5B202_RY601_CV.rValue_OUT;
(* LH601_OP *)
(* LH601_CMD *)
M1_041_5B202_LH601_OP(bPortKNX := 1, dwIndex_DPT := 41, rValue_IN := STLV80_563.STLV80_A_563_5B202.LH601_OP, xUpdate_KNX := i = 9, typDPT := typDPT);
M1_042_5B202_LH601_CMD(bPortKNX := 1, dwIndex_DPT := 42, xSwitch_IN := STLV80_563.STLV80_A_563_5B202.LH601_CMD, xUpdate_KNX := i = 10, typDPT := typDPT);
(* LC601_OP *)
(* LC601_CMD *)
M1_043_5B202_LC601_OP(bPortKNX := 1, dwIndex_DPT := 43, rValue_IN := STLV80_563.STLV80_A_563_5B202.LC601_OP, xUpdate_KNX := i = 11, typDPT := typDPT);
M1_044_5B202_LC601_CMD(bPortKNX := 1, dwIndex_DPT := 44, xSwitch_IN := STLV80_563.STLV80_A_563_5B202.LC601_CMD, xUpdate_KNX := i = 12, typDPT := typDPT);
(* RT601_SP *)
(* RT601_SP Feedback *)
M1_045_5B202_RT601_SP(bPortKNX := 1, dwIndex_DPT := 45, rValue_IN := STLV80_563.STLV80_A_563_5B202.RT601_SP_D, xUpdate_KNX := NOT STLV80_563.STLV80_A_563_5B202.RB601_HVAC, typDPT := typDPT);
M1_046_5B202_RT601_SP_FB(bPortKNX := 1, dwIndex_DPT := 46, typDPT := typDPT);
STLV80_563.STLV80_A_563_5B202.RT601_SP_IN := M1_046_5B202_RT601_SP_FB.rValue_OUT;
(* Rom 5B301 *)
(* RB601_V *)
(* RB601_HVAC *)
M1_047_5B301_RB601_V(bPortKNX := 1, dwIndex_DPT := 47, typDPT := typDPT);
STLV80_563.STLV80_A_563_5B301.RB601_V := M1_047_5B301_RB601_V.xSwitch_OUT;
M1_048_5B301_RB601_HVAC(bPortKNX := 1, dwIndex_DPT := 48, typDPT := typDPT);
STLV80_563.STLV80_A_563_5B301.RB601_HVAC := M1_048_5B301_RB601_HVAC.xSwitch_OUT;
(* RT601_CT *)
(* RY601_CV *)
M1_049_5B301_RT601_CT(bPortKNX := 1, dwIndex_DPT := 49, typDPT := typDPT);
STLV80_563.STLV80_A_563_5B301.RT601_CT := M1_049_5B301_RT601_CT.rValue_OUT;
M1_050_5B301_RY601_CV(bPortKNX := 1, dwIndex_DPT := 50, typDPT := typDPT);
STLV80_563.STLV80_A_563_5B301.RY601_CV := M1_050_5B301_RY601_CV.rValue_OUT;
(* LH601_OP *)
(* LH601_CMD *)
M1_051_5B301_LH601_OP(bPortKNX := 1, dwIndex_DPT := 51, rValue_IN := STLV80_563.STLV80_A_563_5B301.LH601_OP, xUpdate_KNX := i = 13, typDPT := typDPT);
M1_052_5B301_LH601_CMD(bPortKNX := 1, dwIndex_DPT := 52, xSwitch_IN := STLV80_563.STLV80_A_563_5B301.LH601_CMD, xUpdate_KNX := i = 14, typDPT := typDPT);
(* LC601_OP *)
(* LC601_CMD *)
M1_053_5B301_LC601_OP(bPortKNX := 1, dwIndex_DPT := 53, rValue_IN := STLV80_563.STLV80_A_563_5B301.LC601_OP, xUpdate_KNX := i = 15, typDPT := typDPT);
M1_054_5B301_LC601_CMD(bPortKNX := 1, dwIndex_DPT := 54, xSwitch_IN := STLV80_563.STLV80_A_563_5B301.LC601_CMD, xUpdate_KNX := i = 16, typDPT := typDPT);
(* RT601_SP *)
(* RT601_SP Feedback *)
M1_055_5B301_RT601_SP(bPortKNX := 1, dwIndex_DPT := 55, rValue_IN := STLV80_563.STLV80_A_563_5B301.RT601_SP_D, xUpdate_KNX := NOT STLV80_563.STLV80_A_563_5B301.RB601_HVAC, typDPT := typDPT);
M1_056_5B301_RT601_SP_FB(bPortKNX := 1, dwIndex_DPT := 56, typDPT := typDPT);
STLV80_563.STLV80_A_563_5B301.RT601_SP_IN := M1_056_5B301_RT601_SP_FB.rValue_OUT;
(* LU601_V *)
M1_057_5B301_LU601_V(bPortKNX := 1, dwIndex_DPT := 57, typDPT := typDPT);
STLV80_563.STLV80_A_563_5B301.LU601_V := M1_057_5B301_LU601_V.xSwitch_OUT;
(* Rom 5B302 *)
(* RB601_V *)
(* RB601_HVAC *)
M1_058_5B302_RB601_V(bPortKNX := 1, dwIndex_DPT := 58, typDPT := typDPT);
STLV80_563.STLV80_A_563_5B302.RB601_V := M1_058_5B302_RB601_V.xSwitch_OUT;
M1_059_5B302_RB601_HVAC(bPortKNX := 1, dwIndex_DPT := 59, typDPT := typDPT);
STLV80_563.STLV80_A_563_5B302.RB601_HVAC := M1_059_5B302_RB601_HVAC.xSwitch_OUT;
(* RT601_CT *)
(* RY601_CV *)
M1_060_5B302_RT601_CT(bPortKNX := 1, dwIndex_DPT := 60, typDPT := typDPT);
STLV80_563.STLV80_A_563_5B302.RT601_CT := M1_060_5B302_RT601_CT.rValue_OUT;
M1_061_5B302_RY601_CV(bPortKNX := 1, dwIndex_DPT := 61, typDPT := typDPT);
STLV80_563.STLV80_A_563_5B302.RY601_CV := M1_061_5B302_RY601_CV.rValue_OUT;
(* LH601_OP *)
(* LH601_CMD *)
M1_062_5B302_LH601_OP(bPortKNX := 1, dwIndex_DPT := 62, rValue_IN := STLV80_563.STLV80_A_563_5B302.LH601_OP, xUpdate_KNX := i = 17, typDPT := typDPT);
M1_063_5B302_LH601_CMD(bPortKNX := 1, dwIndex_DPT := 63, xSwitch_IN := STLV80_563.STLV80_A_563_5B302.LH601_CMD, xUpdate_KNX := i = 18, typDPT := typDPT);
(* LC601_OP *)
(* LC601_CMD *)
M1_064_5B302_LC601_OP(bPortKNX := 1, dwIndex_DPT := 64, rValue_IN := STLV80_563.STLV80_A_563_5B302.LC601_OP, xUpdate_KNX := i = 19, typDPT := typDPT);
M1_065_5B302_LC601_CMD(bPortKNX := 1, dwIndex_DPT := 65, xSwitch_IN := STLV80_563.STLV80_A_563_5B302.LC601_CMD, xUpdate_KNX := i = 20, typDPT := typDPT);
(* RT601_SP *)
(* RT601_SP Feedback *)
M1_066_5B302_RT601_SP(bPortKNX := 1, dwIndex_DPT := 66, rValue_IN := STLV80_563.STLV80_A_563_5B302.RT601_SP_D, xUpdate_KNX := NOT STLV80_563.STLV80_A_563_5B302.RB601_HVAC, typDPT := typDPT);
M1_067_5B302_RT601_SP_FB(bPortKNX := 1, dwIndex_DPT := 67, typDPT := typDPT);
STLV80_563.STLV80_A_563_5B302.RT601_SP_IN := M1_067_5B302_RT601_SP_FB.rValue_OUT;
(* LU601_V *)
(* LU601_AL *)
M1_068_5B302_LU601_V(bPortKNX := 1, dwIndex_DPT := 68, typDPT := typDPT);
STLV80_563.STLV80_A_563_5B302.LU601_V := M1_068_5B302_LU601_V.xSwitch_OUT;
M1_069_5B302_LU601_AL(bPortKNX := 1, dwIndex_DPT := 69, typDPT := typDPT);
STLV80_563.STLV80_A_563_5B302.LU601_AL := M1_069_5B302_LU601_AL.xSwitch_OUT;
(* Rom 5C201 *)
(* RB601_V *)
(* RB601_HVAC *)
M1_070_5C201_RB601_V(bPortKNX := 1, dwIndex_DPT := 70, typDPT := typDPT);
STLV80_563.STLV80_A_563_5C201.RB601_V := M1_070_5C201_RB601_V.xSwitch_OUT;
M1_071_5C201_RB601_HVAC(bPortKNX := 1, dwIndex_DPT := 71, typDPT := typDPT);
STLV80_563.STLV80_A_563_5C201.RB601_HVAC := M1_071_5C201_RB601_HVAC.xSwitch_OUT;
(* RT601_CT *)
(* RY601_CV *)
M1_072_5C201_RT601_CT(bPortKNX := 1, dwIndex_DPT := 72, typDPT := typDPT);
STLV80_563.STLV80_A_563_5C201.RT601_CT := M1_072_5C201_RT601_CT.rValue_OUT;
M1_073_5C201_RY601_CV(bPortKNX := 1, dwIndex_DPT := 73, typDPT := typDPT);
STLV80_563.STLV80_A_563_5C201.RY601_CV := M1_073_5C201_RY601_CV.rValue_OUT;
(* LH601_OP *)
(* LH601_CMD *)
M1_074_5C201_LH601_OP(bPortKNX := 1, dwIndex_DPT := 74, rValue_IN := STLV80_563.STLV80_A_563_5C201.LH601_OP, xUpdate_KNX := i = 21, typDPT := typDPT);
M1_075_5C201_LH601_CMD(bPortKNX := 1, dwIndex_DPT := 75, xSwitch_IN := STLV80_563.STLV80_A_563_5C201.LH601_CMD, xUpdate_KNX := i = 22, typDPT := typDPT);
(* LC601_OP *)
(* LC601_CMD *)
M1_076_5C201_LC601_OP(bPortKNX := 1, dwIndex_DPT := 76, rValue_IN := STLV80_563.STLV80_A_563_5C201.LC601_OP, xUpdate_KNX := i = 23, typDPT := typDPT);
M1_077_5C201_LC601_CMD(bPortKNX := 1, dwIndex_DPT := 77, xSwitch_IN := STLV80_563.STLV80_A_563_5C201.LC601_CMD, xUpdate_KNX := i = 24, typDPT := typDPT);
(* RT601_SP *)
(* RT601_SP Feedback *)
M1_078_5C201_RT601_SP(bPortKNX := 1, dwIndex_DPT := 78, rValue_IN := STLV80_563.STLV80_A_563_5C201.RT601_SP_D, xUpdate_KNX := NOT STLV80_563.STLV80_A_563_5C201.RB601_HVAC, typDPT := typDPT);
M1_079_5C201_RT601_SP_FB(bPortKNX := 1, dwIndex_DPT := 79, typDPT := typDPT);
STLV80_563.STLV80_A_563_5C201.RT601_SP_IN := M1_079_5C201_RT601_SP_FB.rValue_OUT;
(* LU601_V *)
(* LU601_AL *)
M1_080_5C201_LU601_V(bPortKNX := 1, dwIndex_DPT := 80, typDPT := typDPT);
STLV80_563.STLV80_A_563_5C201.LU601_V := M1_080_5C201_LU601_V.xSwitch_OUT;
M1_081_5C201_LU601_AL(bPortKNX := 1, dwIndex_DPT := 81, typDPT := typDPT);
STLV80_563.STLV80_A_563_5C201.LU601_AL := M1_081_5C201_LU601_AL.xSwitch_OUT;
(* LU601_CMD *)
M1_082_5C201_LU601_CMD(bPortKNX := 1, dwIndex_DPT := 82, xSwitch_IN := STLV80_563.STLV80_A_563_5C201.LU601_CMD, xUpdate_KNX := i = 25, typDPT := typDPT);
(* Rom 5C202 *)
(* RB601_V *)
(* RB602_V *)
M1_083_5C202_RB601_V(bPortKNX := 1, dwIndex_DPT := 83, typDPT := typDPT);
STLV80_563.STLV80_A_563_5C202.RB601_V := M1_083_5C202_RB601_V.xSwitch_OUT;
M1_084_5C202_RB602_V(bPortKNX := 1, dwIndex_DPT := 84, typDPT := typDPT);
STLV80_563.STLV80_A_563_5C202.RB602_V := M1_084_5C202_RB602_V.xSwitch_OUT;
(* RB601_HVAC *)
(* RB602_HVAC *)
M1_085_5C202_RB601_HVAC(bPortKNX := 1, dwIndex_DPT := 85, typDPT := typDPT);
STLV80_563.STLV80_A_563_5C202.RB601_HVAC := M1_085_5C202_RB601_HVAC.xSwitch_OUT;
M1_086_5C202_RB602_HVAC(bPortKNX := 1, dwIndex_DPT := 86, typDPT := typDPT);
STLV80_563.STLV80_A_563_5C202.RB602_HVAC := M1_086_5C202_RB602_HVAC.xSwitch_OUT;
(* RT601_CT *)
(* RT602_CT *)
M1_087_5C202_RT601_CT(bPortKNX := 1, dwIndex_DPT := 87, typDPT := typDPT);
STLV80_563.STLV80_A_563_5C202.RT601_CT := M1_087_5C202_RT601_CT.rValue_OUT;
M1_088_5C202_RT602_CT(bPortKNX := 1, dwIndex_DPT := 88, typDPT := typDPT);
STLV80_563.STLV80_A_563_5C202.RT602_CT := M1_088_5C202_RT602_CT.rValue_OUT;
(* RY601_CV *)
(* RY602_CV *)
M1_089_5C202_RY601_CV(bPortKNX := 1, dwIndex_DPT := 89, typDPT := typDPT);
STLV80_563.STLV80_A_563_5C202.RY601_CV := M1_089_5C202_RY601_CV.rValue_OUT;
M1_090_5C202_RY602_CV(bPortKNX := 1, dwIndex_DPT := 90, typDPT := typDPT);
STLV80_563.STLV80_A_563_5C202.RY602_CV := M1_090_5C202_RY602_CV.rValue_OUT;
(* LH601_OP *)
(* LH602_OP *)
M1_091_5C202_LH601_OP(bPortKNX := 1, dwIndex_DPT := 91, rValue_IN := STLV80_563.STLV80_A_563_5C202.LH601_OP, xUpdate_KNX := i = 26, typDPT := typDPT);
M1_092_5C202_LH602_OP(bPortKNX := 1, dwIndex_DPT := 92, rValue_IN := STLV80_563.STLV80_A_563_5C202.LH602_OP, xUpdate_KNX := i = 27, typDPT := typDPT);
(* LH601_CMD *)
(* LH602_CMD *)
M1_093_5C202_LH601_CMD(bPortKNX := 1, dwIndex_DPT := 93, xSwitch_IN := STLV80_563.STLV80_A_563_5C202.LH601_CMD, xUpdate_KNX := i = 28, typDPT := typDPT);
M1_094_5C202_LH602_CMD(bPortKNX := 1, dwIndex_DPT := 94, xSwitch_IN := STLV80_563.STLV80_A_563_5C202.LH602_CMD, xUpdate_KNX := i = 29, typDPT := typDPT);
(* LC601_OP *)
(* LC602_OP *)
M1_095_5C202_LC601_OP(bPortKNX := 1, dwIndex_DPT := 95, rValue_IN := STLV80_563.STLV80_A_563_5C202.LC601_OP, xUpdate_KNX := i = 30, typDPT := typDPT);
M1_096_5C202_LC602_OP(bPortKNX := 1, dwIndex_DPT := 96, rValue_IN := STLV80_563.STLV80_A_563_5C202.LC602_OP, xUpdate_KNX := i = 31, typDPT := typDPT);
(* LC601_CMD *)
(* LC602_CMD *)
M1_097_5C202_LC601_CMD(bPortKNX := 1, dwIndex_DPT := 97, xSwitch_IN := STLV80_563.STLV80_A_563_5C202.LC601_CMD, xUpdate_KNX := i = 32, typDPT := typDPT);
M1_098_5C202_LC602_CMD(bPortKNX := 1, dwIndex_DPT := 98, xSwitch_IN := STLV80_563.STLV80_A_563_5C202.LC602_CMD, xUpdate_KNX := i = 33, typDPT := typDPT);
(* RT601_SP *)
(* RT602_SP *)
M1_099_5C202_RT601_SP(bPortKNX := 1, dwIndex_DPT := 99, rValue_IN := STLV80_563.STLV80_A_563_5C202.RT601_SP_D, xUpdate_KNX := NOT STLV80_563.STLV80_A_563_5C202.RB601_HVAC, typDPT := typDPT);
M1_0100_5C202_RT602_SP(bPortKNX := 1, dwIndex_DPT := 100, rValue_IN := STLV80_563.STLV80_A_563_5C202.RT602_SP, xUpdate_KNX := NOT STLV80_563.STLV80_A_563_5C202.RB601_HVAC, typDPT := typDPT);
(* RT601_SP Feedback *)
(* RT602_SP Feedback *)
M1_101_5C202_RT601_SP_FB(bPortKNX := 1, dwIndex_DPT := 101, typDPT := typDPT);
STLV80_563.STLV80_A_563_5C202.RT601_SP_IN := M1_101_5C202_RT601_SP_FB.rValue_OUT;
M1_102_5C202_RT602_SP_FB(bPortKNX := 1, dwIndex_DPT := 102, typDPT := typDPT);
STLV80_563.STLV80_A_563_5C202.RT602_SP_IN := M1_102_5C202_RT602_SP_FB.rValue_OUT;
(* LU601_V *)
(* LU602_V *)
M1_103_5C202_LU601_V(bPortKNX := 1, dwIndex_DPT := 103, typDPT := typDPT);
STLV80_563.STLV80_A_563_5C202.LU601_V := M1_103_5C202_LU601_V.xSwitch_OUT;
M1_104_5C202_LU602_V(bPortKNX := 1, dwIndex_DPT := 104, typDPT := typDPT);
STLV80_563.STLV80_A_563_5C202.LU602_V := M1_104_5C202_LU602_V.xSwitch_OUT;
(* LU601_AL *)
(* LU602_AL *)
M1_105_5C202_LU601_AL(bPortKNX := 1, dwIndex_DPT := 105, typDPT := typDPT);
STLV80_563.STLV80_A_563_5C202.LU601_AL := M1_105_5C202_LU601_AL.xSwitch_OUT;
M1_106_5C202_LU602_AL(bPortKNX := 1, dwIndex_DPT := 106, typDPT := typDPT);
STLV80_563.STLV80_A_563_5C202.LU602_AL := M1_106_5C202_LU602_AL.xSwitch_OUT;
(* LU601_CMD *)
(* LU602_CMD *)
M1_107_5C202_LU601_CMD(bPortKNX := 1, dwIndex_DPT := 107, xSwitch_IN := STLV80_563.STLV80_A_563_5C202.LU601_CMD, xUpdate_KNX := i = 34, typDPT := typDPT);
M1_108_5C202_LU602_CMD(bPortKNX := 1, dwIndex_DPT := 108, xSwitch_IN := STLV80_563.STLV80_A_563_5C202.LU602_CMD, xUpdate_KNX := i = 35, typDPT := typDPT);
END_PROGRAM

PROGRAM PRG_563_Romstyring
  VAR
    Rom_5A201 : fbRomtype_112;  (* 5A201 *)
    Rom_5A202 : fbRomtype_11102;  (* 5A202 *)
    Rom_5A203 : fbRomtype_22111;  (* 5A203 *)
    Rom_5A301 : fbRomtype_2211111;  (* 5A301 *)
    Rom_5A302 : fbRomtype_11111111;  (* 5A302 *)
    Rom_5B201 : fbRomtype_111111111;  (* 5B201 *)
    Rom_5B202 : fbRomtype_1111111111;  (* 5B202 *)
    Rom_5B301 : fbRomtype_11111111111;  (* 5B301 *)
    Rom_5B302 : fbRomtype_111111111111;  (* 5B302 *)
    Rom_5C201 : fbRomtype_1111111111111;  (* 5C201 *)
    Rom_5C202 : fbRomtype_2222222222222;  (* 5C202 *)
  END_VAR

(* CFC diagram, written out as Structured Text *)
(* Rom 5A201 *)
Rom_5A201(RB601_HVAC := STLV80_563.STLV80_A_563_5A201.RB601_HVAC, RT601_CT := STLV80_563.STLV80_A_563_5A201.RT601_CT, RT602_CT := STLV80_563.STLV80_A_563_5A201.RT602_CT, RT602_SP := STLV80_563.STLV80_A_563_5A201.RT602_SP, RT601_SP_D := STLV80_563.STLV80_A_563_5A201.RT601_SP_D, RT601_SP_S := STLV80_563.STLV80_A_563_5A201.RT601_SP_S, RT601_SP_N := STLV80_563.STLV80_A_563_5A201.RT601_SP_N, RT601_SP_F := STLV80_563.STLV80_A_563_5A201.RT601_SP_F, OPM := STLV80_563.STLV80_A_563_5A201.OPM);
STLV80_563.STLV80_A_563_5A201.OPM_CV := Rom_5A201.OPM_CV;
STLV80_563.STLV80_A_563_5A201.RT601_CS := Rom_5A201.RT601_CS;
(* Rom 5A202 *)
Rom_5A202(RB601_HVAC := STLV80_563.STLV80_A_563_5A202.RB601_HVAC, RT601_CT := STLV80_563.STLV80_A_563_5A202.RT601_CT, RT601_SP_D := STLV80_563.STLV80_A_563_5A202.RT601_SP_D, RT601_SP_S := STLV80_563.STLV80_A_563_5A202.RT601_SP_S, RT601_SP_N := STLV80_563.STLV80_A_563_5A202.RT601_SP_N, RT601_SP_F := STLV80_563.STLV80_A_563_5A202.RT601_SP_F, OPM := STLV80_563.STLV80_A_563_5A202.OPM, LH601_MAN := STLV80_563.STLV80_A_563_5A202.LH601_MAN);
STLV80_563.STLV80_A_563_5A202.OPM_CV := Rom_5A202.OPM_CV;
STLV80_563.STLV80_A_563_5A202.RT601_CS := Rom_5A202.RT601_CS;
STLV80_563.STLV80_A_563_5A202.LH601_OP := Rom_5A202.LH601_OP;
STLV80_563.STLV80_A_563_5A202.LH602_OP := Rom_5A202.LH602_OP;
(* Rom 5A203 *)
Rom_5A203(RB601_HVAC := STLV80_563.STLV80_A_563_5A203.RB601_HVAC, RB602_HVAC := STLV80_563.STLV80_A_563_5A203.RB602_HVAC, RT601_CT := STLV80_563.STLV80_A_563_5A203.RT601_CT, RT601_SP_D := STLV80_563.STLV80_A_563_5A203.RT601_SP_D, RT601_SP_S := STLV80_563.STLV80_A_563_5A203.RT601_SP_S, RT601_SP_N := STLV80_563.STLV80_A_563_5A203.RT601_SP_N, RT601_SP_F := STLV80_563.STLV80_A_563_5A203.RT601_SP_F, OPM := STLV80_563.STLV80_A_563_5A203.OPM, RY601_CV := STLV80_563.STLV80_A_563_5A203.RY601_CV, RY601_SP := STLV80_563.STLV80_A_563_5A203.RY601_SP, LH601_MAN := STLV80_563.STLV80_A_563_5A203.LH601_MAN);
STLV80_563.STLV80_A_563_5A203.OPM_CV := Rom_5A203.OPM_CV;
STLV80_563.STLV80_A_563_5A203.RT601_CS := Rom_5A203.RT601_CS;
STLV80_563.STLV80_A_563_5A203.RY601_OP := Rom_5A203.RY601_OP;
STLV80_563.STLV80_A_563_5A203.LH601_OP := Rom_5A203.LH601_OP;
(* Rom 5A301 *)
Rom_5A301(RB601_HVAC := STLV80_563.STLV80_A_563_5A301.RB601_HVAC, RB602_HVAC := STLV80_563.STLV80_A_563_5A301.RB602_HVAC, RT601_CT := STLV80_563.STLV80_A_563_5A301.RT601_CT, RT601_SP_D := STLV80_563.STLV80_A_563_5A301.RT601_SP_D, RT601_SP_S := STLV80_563.STLV80_A_563_5A301.RT601_SP_S, RT601_SP_N := STLV80_563.STLV80_A_563_5A301.RT601_SP_N, RT601_SP_F := STLV80_563.STLV80_A_563_5A301.RT601_SP_F, OPM := STLV80_563.STLV80_A_563_5A301.OPM, RY601_CV := STLV80_563.STLV80_A_563_5A301.RY601_CV, RY601_SP := STLV80_563.STLV80_A_563_5A301.RY601_SP, LH601_MAN := STLV80_563.STLV80_A_563_5A301.LH601_MAN, LC601_MAN := STLV80_563.STLV80_A_563_5A301.LC601_MAN);
STLV80_563.STLV80_A_563_5A301.OPM_CV := Rom_5A301.OPM_CV;
STLV80_563.STLV80_A_563_5A301.RT601_CS := Rom_5A301.RT601_CS;
STLV80_563.STLV80_A_563_5A301.RY601_OP := Rom_5A301.RY601_OP;
STLV80_563.STLV80_A_563_5A301.LH601_OP := Rom_5A301.LH601_OP;
STLV80_563.STLV80_A_563_5A301.LH601_CMD := Rom_5A301.LH601_CMD;
STLV80_563.STLV80_A_563_5A301.LC601_OP := Rom_5A301.LC601_OP;
(* Rom 5A302 *)
Rom_5A302(RB601_HVAC := STLV80_563.STLV80_A_563_5A302.RB601_HVAC, RT601_CT := STLV80_563.STLV80_A_563_5A302.RT601_CT, RT601_SP_D := STLV80_563.STLV80_A_563_5A302.RT601_SP_D, RT601_SP_S := STLV80_563.STLV80_A_563_5A302.RT601_SP_S, RT601_SP_N := STLV80_563.STLV80_A_563_5A302.RT601_SP_N, RT601_SP_F := STLV80_563.STLV80_A_563_5A302.RT601_SP_F, OPM := STLV80_563.STLV80_A_563_5A302.OPM, RY601_CV := STLV80_563.STLV80_A_563_5A302.RY601_CV, RY601_SP := STLV80_563.STLV80_A_563_5A302.RY601_SP, LH601_MAN := STLV80_563.STLV80_A_563_5A302.LH601_MAN, LC601_MAN := STLV80_563.STLV80_A_563_5A302.LC601_MAN);
STLV80_563.STLV80_A_563_5A302.OPM_CV := Rom_5A302.OPM_CV;
STLV80_563.STLV80_A_563_5A302.RT601_CS := Rom_5A302.RT601_CS;
STLV80_563.STLV80_A_563_5A302.RY601_OP := Rom_5A302.RY601_OP;
STLV80_563.STLV80_A_563_5A302.LH601_OP := Rom_5A302.LH601_OP;
STLV80_563.STLV80_A_563_5A302.LH601_CMD := Rom_5A302.LH601_CMD;
STLV80_563.STLV80_A_563_5A302.LC601_OP := Rom_5A302.LC601_OP;
STLV80_563.STLV80_A_563_5A302.LC601_CMD := Rom_5A302.LC601_CMD;
(* Rom 5B201 *)
Rom_5B201(RB601_HVAC := STLV80_563.STLV80_A_563_5B201.RB601_HVAC, RT601_CT := STLV80_563.STLV80_A_563_5B201.RT601_CT, RT601_SP_D := STLV80_563.STLV80_A_563_5B201.RT601_SP_D, RT601_SP_S := STLV80_563.STLV80_A_563_5B201.RT601_SP_S, RT601_SP_N := STLV80_563.STLV80_A_563_5B201.RT601_SP_N, RT601_SP_F := STLV80_563.STLV80_A_563_5B201.RT601_SP_F, OPM := STLV80_563.STLV80_A_563_5B201.OPM, RY601_CV := STLV80_563.STLV80_A_563_5B201.RY601_CV, RY601_SP := STLV80_563.STLV80_A_563_5B201.RY601_SP, LH601_MAN := STLV80_563.STLV80_A_563_5B201.LH601_MAN, LC601_MAN := STLV80_563.STLV80_A_563_5B201.LC601_MAN);
STLV80_563.STLV80_A_563_5B201.OPM_CV := Rom_5B201.OPM_CV;
STLV80_563.STLV80_A_563_5B201.RT601_CS := Rom_5B201.RT601_CS;
STLV80_563.STLV80_A_563_5B201.RY601_OP := Rom_5B201.RY601_OP;
STLV80_563.STLV80_A_563_5B201.LH601_OP := Rom_5B201.LH601_OP;
STLV80_563.STLV80_A_563_5B201.LH601_CMD := Rom_5B201.LH601_CMD;
STLV80_563.STLV80_A_563_5B201.LC601_OP := Rom_5B201.LC601_OP;
STLV80_563.STLV80_A_563_5B201.LC601_CMD := Rom_5B201.LC601_CMD;
(* Rom 5B202 *)
Rom_5B202(RB601_HVAC := STLV80_563.STLV80_A_563_5B202.RB601_HVAC, RT601_CT := STLV80_563.STLV80_A_563_5B202.RT601_CT, RT601_SP_D := STLV80_563.STLV80_A_563_5B202.RT601_SP_D, RT601_SP_S := STLV80_563.STLV80_A_563_5B202.RT601_SP_S, RT601_SP_N := STLV80_563.STLV80_A_563_5B202.RT601_SP_N, RT601_SP_F := STLV80_563.STLV80_A_563_5B202.RT601_SP_F, OPM := STLV80_563.STLV80_A_563_5B202.OPM, RY601_CV := STLV80_563.STLV80_A_563_5B202.RY601_CV, RY601_SP := STLV80_563.STLV80_A_563_5B202.RY601_SP, LH601_MAN := STLV80_563.STLV80_A_563_5B202.LH601_MAN, LC601_MAN := STLV80_563.STLV80_A_563_5B202.LC601_MAN);
STLV80_563.STLV80_A_563_5B202.OPM_CV := Rom_5B202.OPM_CV;
STLV80_563.STLV80_A_563_5B202.RT601_CS := Rom_5B202.RT601_CS;
STLV80_563.STLV80_A_563_5B202.RY601_OP := Rom_5B202.RY601_OP;
STLV80_563.STLV80_A_563_5B202.LH601_OP := Rom_5B202.LH601_OP;
STLV80_563.STLV80_A_563_5B202.LH601_CMD := Rom_5B202.LH601_CMD;
STLV80_563.STLV80_A_563_5B202.LC601_OP := Rom_5B202.LC601_OP;
STLV80_563.STLV80_A_563_5B202.LC601_CMD := Rom_5B202.LC601_CMD;
(* Rom 5B301 *)
Rom_5B301(RB601_HVAC := STLV80_563.STLV80_A_563_5B301.RB601_HVAC, RT601_CT := STLV80_563.STLV80_A_563_5B301.RT601_CT, RT601_SP_D := STLV80_563.STLV80_A_563_5B301.RT601_SP_D, RT601_SP_S := STLV80_563.STLV80_A_563_5B301.RT601_SP_S, RT601_SP_N := STLV80_563.STLV80_A_563_5B301.RT601_SP_N, RT601_SP_F := STLV80_563.STLV80_A_563_5B301.RT601_SP_F, OPM := STLV80_563.STLV80_A_563_5B301.OPM, RY601_CV := STLV80_563.STLV80_A_563_5B301.RY601_CV, RY601_SP := STLV80_563.STLV80_A_563_5B301.RY601_SP, LH601_MAN := STLV80_563.STLV80_A_563_5B301.LH601_MAN, LC601_MAN := STLV80_563.STLV80_A_563_5B301.LC601_MAN, RT601_SP_IN := STLV80_563.STLV80_A_563_5B301.RT601_SP_IN);
STLV80_563.STLV80_A_563_5B301.OPM_CV := Rom_5B301.OPM_CV;
STLV80_563.STLV80_A_563_5B301.RT601_CS := Rom_5B301.RT601_CS;
STLV80_563.STLV80_A_563_5B301.RY601_OP := Rom_5B301.RY601_OP;
STLV80_563.STLV80_A_563_5B301.LH601_OP := Rom_5B301.LH601_OP;
STLV80_563.STLV80_A_563_5B301.LH601_CMD := Rom_5B301.LH601_CMD;
STLV80_563.STLV80_A_563_5B301.LC601_OP := Rom_5B301.LC601_OP;
STLV80_563.STLV80_A_563_5B301.LC601_CMD := Rom_5B301.LC601_CMD;
(* Rom 5B302 *)
Rom_5B302(RB601_HVAC := STLV80_563.STLV80_A_563_5B302.RB601_HVAC, RT601_CT := STLV80_563.STLV80_A_563_5B302.RT601_CT, RT601_SP_D := STLV80_563.STLV80_A_563_5B302.RT601_SP_D, RT601_SP_S := STLV80_563.STLV80_A_563_5B302.RT601_SP_S, RT601_SP_N := STLV80_563.STLV80_A_563_5B302.RT601_SP_N, RT601_SP_F := STLV80_563.STLV80_A_563_5B302.RT601_SP_F, OPM := STLV80_563.STLV80_A_563_5B302.OPM, RY601_CV := STLV80_563.STLV80_A_563_5B302.RY601_CV, RY601_SP := STLV80_563.STLV80_A_563_5B302.RY601_SP, LH601_MAN := STLV80_563.STLV80_A_563_5B302.LH601_MAN, LC601_MAN := STLV80_563.STLV80_A_563_5B302.LC601_MAN, RT601_SP_IN := STLV80_563.STLV80_A_563_5B302.RT601_SP_IN, LU601_V := STLV80_563.STLV80_A_563_5B302.LU601_V);
STLV80_563.STLV80_A_563_5B302.OPM_CV := Rom_5B302.OPM_CV;
STLV80_563.STLV80_A_563_5B302.RT601_CS := Rom_5B302.RT601_CS;
STLV80_563.STLV80_A_563_5B302.RY601_OP := Rom_5B302.RY601_OP;
STLV80_563.STLV80_A_563_5B302.LH601_OP := Rom_5B302.LH601_OP;
STLV80_563.STLV80_A_563_5B302.LH601_CMD := Rom_5B302.LH601_CMD;
STLV80_563.STLV80_A_563_5B302.LC601_OP := Rom_5B302.LC601_OP;
STLV80_563.STLV80_A_563_5B302.LC601_CMD := Rom_5B302.LC601_CMD;
(* Rom 5C201 *)
Rom_5C201(RB601_HVAC := STLV80_563.STLV80_A_563_5C201.RB601_HVAC, RT601_CT := STLV80_563.STLV80_A_563_5C201.RT601_CT, RT601_SP_D := STLV80_563.STLV80_A_563_5C201.RT601_SP_D, RT601_SP_S := STLV80_563.STLV80_A_563_5C201.RT601_SP_S, RT601_SP_N := STLV80_563.STLV80_A_563_5C201.RT601_SP_N, RT601_SP_F := STLV80_563.STLV80_A_563_5C201.RT601_SP_F, OPM := STLV80_563.STLV80_A_563_5C201.OPM, RY601_CV := STLV80_563.STLV80_A_563_5C201.RY601_CV, RY601_SP := STLV80_563.STLV80_A_563_5C201.RY601_SP, LH601_MAN := STLV80_563.STLV80_A_563_5C201.LH601_MAN, LC601_MAN := STLV80_563.STLV80_A_563_5C201.LC601_MAN, RT601_SP_IN := STLV80_563.STLV80_A_563_5C201.RT601_SP_IN, LU601_V := STLV80_563.STLV80_A_563_5C201.LU601_V);
STLV80_563.STLV80_A_563_5C201.OPM_CV := Rom_5C201.OPM_CV;
STLV80_563.STLV80_A_563_5C201.RT601_CS := Rom_5C201.RT601_CS;
STLV80_563.STLV80_A_563_5C201.RY601_OP := Rom_5C201.RY601_OP;
STLV80_563.STLV80_A_563_5C201.LH601_OP := Rom_5C201.LH601_OP;
STLV80_563.STLV80_A_563_5C201.LH601_CMD := Rom_5C201.LH601_CMD;
STLV80_563.STLV80_A_563_5C201.LC601_OP := Rom_5C201.LC601_OP;
STLV80_563.STLV80_A_563_5C201.LC601_CMD := Rom_5C201.LC601_CMD;
STLV80_563.STLV80_A_563_5C201.LU601_CMD := Rom_5C201.LU601_CMD;
(* Rom 5C202 *)
Rom_5C202(RB601_HVAC := STLV80_563.STLV80_A_563_5C202.RB601_HVAC, RB602_HVAC := STLV80_563.STLV80_A_563_5C202.RB602_HVAC, RT601_CT := STLV80_563.STLV80_A_563_5C202.RT601_CT, RT602_CT := STLV80_563.STLV80_A_563_5C202.RT602_CT, RT602_SP := STLV80_563.STLV80_A_563_5C202.RT602_SP, RT601_SP_D := STLV80_563.STLV80_A_563_5C202.RT601_SP_D, RT601_SP_S := STLV80_563.STLV80_A_563_5C202.RT601_SP_S, RT601_SP_N := STLV80_563.STLV80_A_563_5C202.RT601_SP_N, RT601_SP_F := STLV80_563.STLV80_A_563_5C202.RT601_SP_F, OPM := STLV80_563.STLV80_A_563_5C202.OPM, RY601_CV := STLV80_563.STLV80_A_563_5C202.RY601_CV, RY602_CV := STLV80_563.STLV80_A_563_5C202.RY602_CV, RY601_SP := STLV80_563.STLV80_A_563_5C202.RY601_SP, LH601_MAN := STLV80_563.STLV80_A_563_5C202.LH601_MAN, LC601_MAN := STLV80_563.STLV80_A_563_5C202.LC601_MAN, RT601_SP_IN := STLV80_563.STLV80_A_563_5C202.RT601_SP_IN, RT602_SP_IN := STLV80_563.STLV80_A_563_5C202.RT602_SP_IN, LU601_V := STLV80_563.STLV80_A_563_5C202.LU601_V, LU602_V := STLV80_563.STLV80_A_563_5C202.LU602_V);
STLV80_563.STLV80_A_563_5C202.OPM_CV := Rom_5C202.OPM_CV;
STLV80_563.STLV80_A_563_5C202.RT601_CS := Rom_5C202.RT601_CS;
STLV80_563.STLV80_A_563_5C202.RY601_OP := Rom_5C202.RY601_OP;
STLV80_563.STLV80_A_563_5C202.LH601_OP := Rom_5C202.LH601_OP;
STLV80_563.STLV80_A_563_5C202.LH602_OP := Rom_5C202.LH602_OP;
STLV80_563.STLV80_A_563_5C202.LH601_CMD := Rom_5C202.LH601_CMD;
STLV80_563.STLV80_A_563_5C202.LH602_CMD := Rom_5C202.LH602_CMD;
STLV80_563.STLV80_A_563_5C202.LC601_OP := Rom_5C202.LC601_OP;
STLV80_563.STLV80_A_563_5C202.LC602_OP := Rom_5C202.LC602_OP;
STLV80_563.STLV80_A_563_5C202.LC601_CMD := Rom_5C202.LC601_CMD;
STLV80_563.STLV80_A_563_5C202.LC602_CMD := Rom_5C202.LC602_CMD;
STLV80_563.STLV80_A_563_5C202.LU601_CMD := Rom_5C202.LU601_CMD;
STLV80_563.STLV80_A_563_5C202.LU602_CMD := Rom_5C202.LU602_CMD;
END_PROGRAM
